// TIA Portal project "analog" (V17)
// Vorlageprojekt für das Buch mit Zielsystem S7-1200

(* hardware
DEVICE "S7-1200-Station_1"  S7-1200 Station
   slot 0: "Baugruppenträger_0"  Rack  V1.0
   slot 1: "PLC_1"  CPU 1211C DC/DC/DC  6ES7 211-1AE40-0XB0  V4.1
*)

// ===== PLC "PLC_1"  CPU 1211C DC/DC/DC =====

VAR_GLOBAL   // PLC tag table "Standard-Variablentabelle"
   "movingX" AT %I0.0 : Bool;
   "movingZ" AT %I0.1 : Bool;
   "itemDetected" AT %I0.2 : Bool;
   "lidAtPLace" AT %I0.3 : Bool;
   "lidClamped" AT %I0.4 : Bool;
   "PosAtLImit(Lids)" AT %I0.5 : Bool;
   "baseAtPlace" AT %I0.6 : Bool;
   "baseClamped" AT %I0.7 : Bool;
   "PosAtLImit(bases)" AT %I1.0 : Bool;
   "partLeaving" AT %I1.1 : Bool;
   "start" AT %I1.2 : Bool;
   "reset" AT %I1.3 : Bool;
   "stop" AT %I1.4 : Bool;
   "emergencyStop" AT %I1.5 : Bool;
   "auto" AT %I1.6 : Bool;
   "factoryIORunning" AT %I1.7 : Bool;
   "moveX" AT %Q0.0 : Bool;
   "moveZ" AT %Q0.1 : Bool;
   "grab" AT %Q0.2 : Bool;
   "lidsConveyor" AT %Q0.3 : Bool;
   "clampLid" AT %Q0.4 : Bool;
   "posRaise(lids)" AT %Q0.5 : Bool;
   "basesConveyor" AT %Q0.6 : Bool;
   "clampBAse" AT %Q0.7 : Bool;
   "posRaise(bases)" AT %Q1.0 : Bool;
   "startLight" AT %Q1.1 : Bool;
   "resetLight" AT %Q1.2 : Bool;
   "stopLight" AT %Q1.3 : Bool;
   "counter" AT %QD30 : DWord;
   "autoMode" AT %M0.0 : Bool;
   "manualMode" AT %M0.1 : Bool;
   "emergencyActivated" AT %M0.2 : Bool;
   "Clock_Byte" AT %MB10 : Byte;
   "Clock_10Hz" AT %M10.0 : Bool;
   "Clock_5Hz" AT %M10.1 : Bool;
   "Clock_2.5Hz" AT %M10.2 : Bool;
   "Clock_2Hz" AT %M10.3 : Bool;
   "Clock_1.25Hz" AT %M10.4 : Bool;
   "Clock_1Hz" AT %M10.5 : Bool;
   "Clock_0.625Hz" AT %M10.6 : Bool;
   "Clock_0.5Hz" AT %M10.7 : Bool;
   "systemRun" AT %M0.3 : Bool;
   "resetMode" AT %M0.4 : Bool;
   "Tag_1" AT %M8.0 : Bool;
   "Tag_2" AT %M8.1 : Bool;
   "Tag_3" AT %M8.2 : Bool;
   "lidAligned" AT %M0.5 : Bool;
   "moveZBit1" AT %M0.6 : Bool;
   "Tag_4" AT %M8.3 : Bool;
   "Tag_5" AT %M8.4 : Bool;
   "initiateStep8" AT %M0.7 : Bool;
   "Tag_6" AT %M8.5 : Bool;
   "Tag_7" AT %M8.6 : Bool;
   "moveZBit2" AT %M1.0 : Bool;
   "Tag_8" AT %M8.7 : Bool;
   "temp1" AT %M1.1 : Bool;
   "temp2" AT %M1.2 : Bool;
   "Tag_9" AT %M9.0 : Bool;
   "Tag_10" AT %M9.2 : Bool;
   "loop" AT %M1.3 : Bool;
END_VAR

DATA_BLOCK "manualCounterCount"   // DB4
{ S7_Optimized_Access := 'TRUE' }
VERSION : 0.1
   VAR
      manualCount : Int := -1;
   END_VAR
BEGIN
END_DATA_BLOCK

// folder: System blocks/Program resources

DATA_BLOCK "timer1"   // DB1
{ S7_Optimized_Access := 'TRUE' }
AUTHOR : Simatic
FAMILY : IEC
NAME : IEC_TMR
VERSION : 1.0
// stored: InstanceOfName IEC_TIMER
"IEC_TIMER"
BEGIN
END_DATA_BLOCK

DATA_BLOCK "timer2"   // DB2
{ S7_Optimized_Access := 'TRUE' }
AUTHOR : Simatic
FAMILY : IEC
NAME : IEC_TMR
VERSION : 1.0
// stored: InstanceOfName IEC_TIMER
"IEC_TIMER"
BEGIN
END_DATA_BLOCK

// folder: (top level)

FUNCTION "modesOf Operation" : Void   // FC1, LAD
{ S7_Optimized_Access := 'TRUE' }
VERSION : 0.1
   VAR_TEMP   // added for the SCL form of the ladder/FBD networks
      _w1 : Bool;
   END_VAR
BEGIN

REGION Network 1: Manual/AutoMode selector switch
   // Switches between manual and automatic modes
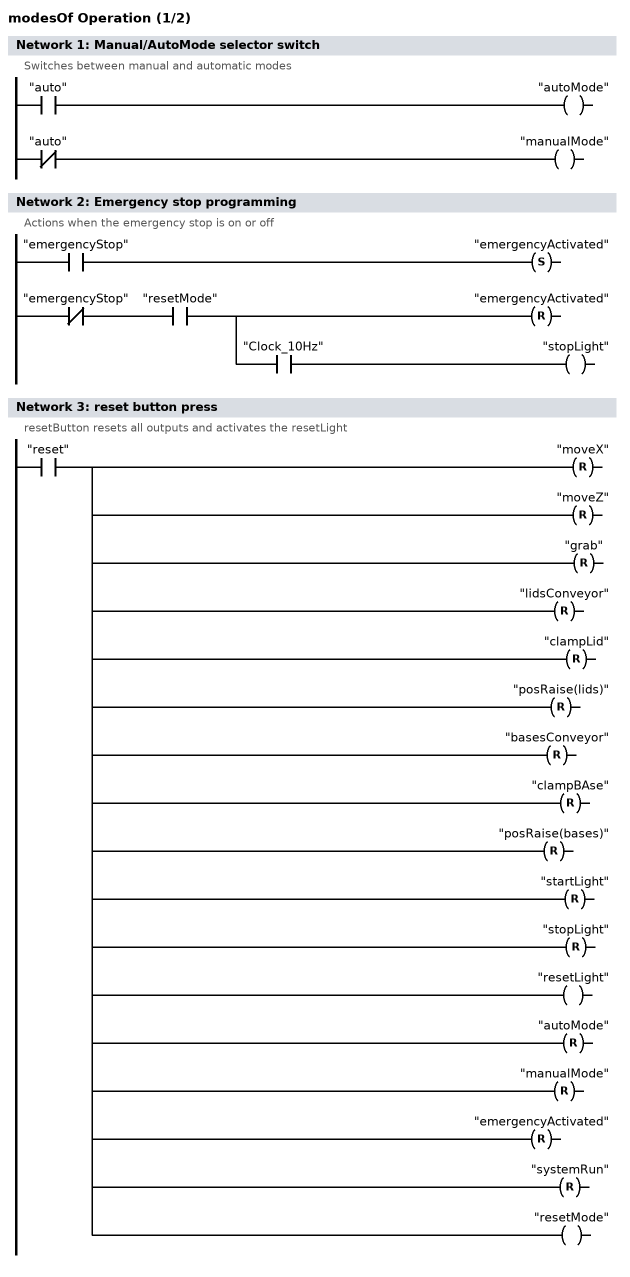
   RUNG wire#powerrail
      Contact( "auto" )
      Coil( "autoMode" )
   END_RUNG
   RUNG wire#powerrail
      I_Contact( "auto" )
      Coil( "manualMode" )
   END_RUNG
   // the same network as SCL:
   "autoMode" := "auto";
   "manualMode" := NOT "auto";
END_REGION

REGION Network 2: Emergency stop programming
   // Actions when the emergency stop is on or off
   RUNG wire#powerrail
      Contact( "emergencyStop" )
      S_Coil( "emergencyActivated" )
   END_RUNG
   RUNG wire#powerrail
      I_Contact( "emergencyStop" )
      Contact( "resetMode" )
      wire#w1
      R_Coil( "emergencyActivated" )
   END_RUNG
   RUNG wire#w1
      Contact( "Clock_10Hz" )
      Coil( "stopLight" )
   END_RUNG
   // the same network as SCL:
   IF "emergencyStop" THEN "emergencyActivated" := TRUE; END_IF;
   #_w1 := NOT "emergencyStop" AND "resetMode";
   IF #_w1 THEN "emergencyActivated" := FALSE; END_IF;
   "stopLight" := #_w1 AND "Clock_10Hz";
END_REGION

REGION Network 3: reset button press
   // resetButton resets all outputs and activates the resetLight
   RUNG wire#powerrail
      Contact( "reset" )
      wire#w1
      R_Coil( "moveX" )
   END_RUNG
   RUNG wire#w1
      R_Coil( "moveZ" )
   END_RUNG
   RUNG wire#w1
      R_Coil( "grab" )
   END_RUNG
   RUNG wire#w1
      R_Coil( "lidsConveyor" )
   END_RUNG
   RUNG wire#w1
      R_Coil( "clampLid" )
   END_RUNG
   RUNG wire#w1
      R_Coil( "posRaise(lids)" )
   END_RUNG
   RUNG wire#w1
      R_Coil( "basesConveyor" )
   END_RUNG
   RUNG wire#w1
      R_Coil( "clampBAse" )
   END_RUNG
   RUNG wire#w1
      R_Coil( "posRaise(bases)" )
   END_RUNG
   RUNG wire#w1
      R_Coil( "startLight" )
   END_RUNG
   RUNG wire#w1
      R_Coil( "stopLight" )
   END_RUNG
   RUNG wire#w1
      Coil( "resetLight" )
   END_RUNG
   RUNG wire#w1
      R_Coil( "autoMode" )
   END_RUNG
   RUNG wire#w1
      R_Coil( "manualMode" )
   END_RUNG
   RUNG wire#w1
      R_Coil( "emergencyActivated" )
   END_RUNG
   RUNG wire#w1
      R_Coil( "systemRun" )
   END_RUNG
   RUNG wire#w1
      Coil( "resetMode" )
   END_RUNG
   // the same network as SCL:
   IF "reset" THEN
       "moveX" := FALSE;
       "moveZ" := FALSE;
       "grab" := FALSE;
       "lidsConveyor" := FALSE;
       "clampLid" := FALSE;
       "posRaise(lids)" := FALSE;
       "basesConveyor" := FALSE;
       "clampBAse" := FALSE;
       "posRaise(bases)" := FALSE;
       "startLight" := FALSE;
       "stopLight" := FALSE;
   END_IF;
   "resetLight" := "reset";
   IF "reset" THEN
       "autoMode" := FALSE;
       "manualMode" := FALSE;
       "emergencyActivated" := FALSE;
       "systemRun" := FALSE;
   END_IF;
   "resetMode" := "reset";
END_REGION

REGION Network 4: Start button press
   // when the start button is pressed it should activate the system should run . Action of the stop and emergency stop should stop the system from working
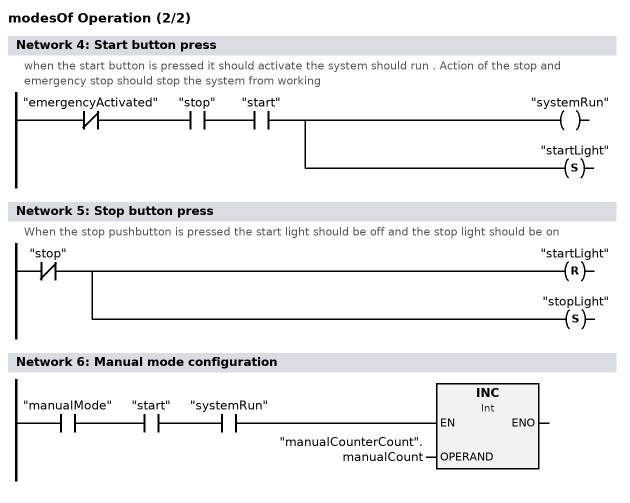
   RUNG wire#powerrail
      I_Contact( "emergencyActivated" )
      Contact( "stop" )
      Contact( "start" )
      wire#w1
      Coil( "systemRun" )
   END_RUNG
   RUNG wire#w1
      S_Coil( "startLight" )
   END_RUNG
   // the same network as SCL:
   "systemRun" := NOT "emergencyActivated" AND "stop" AND "start";
   IF "systemRun" THEN "startLight" := TRUE; END_IF;
END_REGION

REGION Network 5: Stop button press
   // When the stop pushbutton is pressed the start light should be off and the stop light should be on
   RUNG wire#powerrail
      I_Contact( "stop" )
      wire#w1
      R_Coil( "startLight" )
   END_RUNG
   RUNG wire#w1
      S_Coil( "stopLight" )
   END_RUNG
   // the same network as SCL:
   IF NOT "stop" THEN
       "startLight" := FALSE;
       "stopLight" := TRUE;
   END_IF;
END_REGION

REGION Network 6: Manual mode configuration
   RUNG wire#powerrail
      Contact( "manualMode" )
      Contact( "start" )
      Contact( "systemRun" )
      { S7_Templates := "DestType := Int" } Inc( "manualCounterCount".manualCount )
   END_RUNG
   // the same network as SCL:
   IF "manualMode" AND "start" AND "systemRun" THEN
       "manualCounterCount".manualCount := "manualCounterCount".manualCount + 1;
   END_IF;
END_REGION
END_FUNCTION

FUNCTION "stepDfn" : Void   // FC2, LAD
{ S7_Optimized_Access := 'TRUE' }
VERSION : 0.1
   VAR_TEMP   // added for the SCL form of the ladder/FBD networks
      _w1 : Bool;
      _w2 : Bool;
   END_VAR
BEGIN

REGION Network 1: Step 1
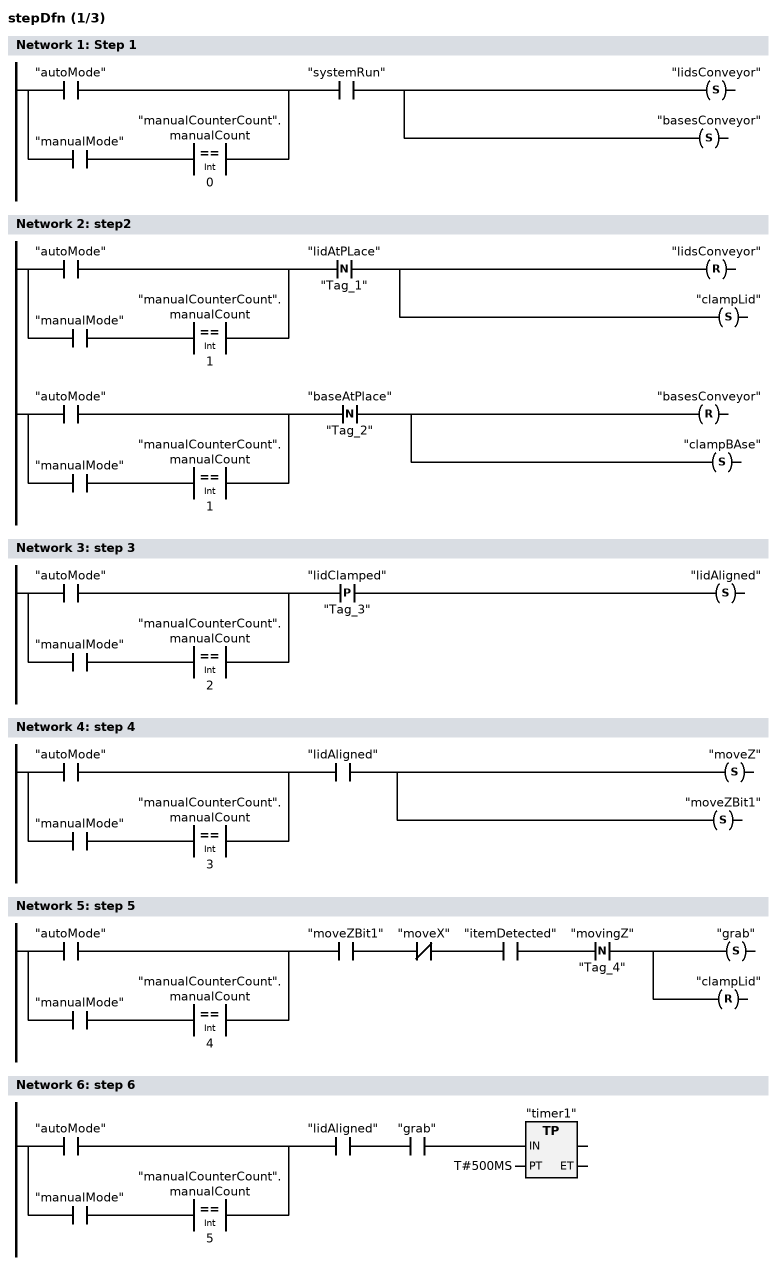
   RUNG wire#powerrail
      Contact( "autoMode" )
      wire#w1
      Contact( "systemRun" )
      wire#w2
      S_Coil( "lidsConveyor" )
   END_RUNG
   RUNG wire#powerrail
      Contact( "manualMode" )
      { S7_Templates := "SrcType := Int" } EQ_Contact(in1 := "manualCounterCount".manualCount, in2 := 0)
   END_RUNG wire#w1
   RUNG wire#w2
      S_Coil( "basesConveyor" )
   END_RUNG
   // the same network as SCL:
   IF ("autoMode" OR ("manualMode" AND ("manualCounterCount".manualCount = 0))) AND "systemRun" THEN
       "lidsConveyor" := TRUE;
       "basesConveyor" := TRUE;
   END_IF;
END_REGION

REGION Network 2: step2
   RUNG wire#powerrail
      Contact( "autoMode" )
      wire#w1
      N_Contact(operand := "lidAtPLace", bit := "Tag_1")
      wire#w2
      R_Coil( "lidsConveyor" )
   END_RUNG
   RUNG wire#powerrail
      Contact( "manualMode" )
      { S7_Templates := "SrcType := Int" } EQ_Contact(in1 := "manualCounterCount".manualCount, in2 := 1)
   END_RUNG wire#w1
   RUNG wire#w2
      S_Coil( "clampLid" )
   END_RUNG
   RUNG wire#powerrail
      Contact( "autoMode" )
      wire#w3
      N_Contact(operand := "baseAtPlace", bit := "Tag_2")
      wire#w4
      R_Coil( "basesConveyor" )
   END_RUNG
   RUNG wire#powerrail
      Contact( "manualMode" )
      { S7_Templates := "SrcType := Int" } EQ_Contact(in1 := "manualCounterCount".manualCount, in2 := 1)
   END_RUNG wire#w3
   RUNG wire#w4
      S_Coil( "clampBAse" )
   END_RUNG
   // the same network as SCL:
   #_w1 := ("autoMode" OR ("manualMode" AND ("manualCounterCount".manualCount = 1))) AND NOT "lidAtPLace" AND "Tag_1";   // falling edge of "lidAtPLace"
   "Tag_1" := "lidAtPLace";
   IF #_w1 THEN
       "lidsConveyor" := FALSE;
       "clampLid" := TRUE;
   END_IF;
   #_w2 := ("autoMode" OR ("manualMode" AND ("manualCounterCount".manualCount = 1))) AND NOT "baseAtPlace" AND "Tag_2";   // falling edge of "baseAtPlace"
   "Tag_2" := "baseAtPlace";
   IF #_w2 THEN
       "basesConveyor" := FALSE;
       "clampBAse" := TRUE;
   END_IF;
END_REGION

REGION Network 3: step 3
   RUNG wire#powerrail
      Contact( "autoMode" )
      wire#w1
      P_Contact(operand := "lidClamped", bit := "Tag_3")
      S_Coil( "lidAligned" )
   END_RUNG
   RUNG wire#powerrail
      Contact( "manualMode" )
      { S7_Templates := "SrcType := Int" } EQ_Contact(in1 := "manualCounterCount".manualCount, in2 := 2)
   END_RUNG wire#w1
   // the same network as SCL:
   #_w1 := ("autoMode" OR ("manualMode" AND ("manualCounterCount".manualCount = 2))) AND "lidClamped" AND NOT "Tag_3";   // rising edge of "lidClamped"
   "Tag_3" := "lidClamped";
   IF #_w1 THEN "lidAligned" := TRUE; END_IF;
END_REGION

REGION Network 4: step 4
   RUNG wire#powerrail
      Contact( "autoMode" )
      wire#w1
      Contact( "lidAligned" )
      wire#w2
      S_Coil( "moveZ" )
   END_RUNG
   RUNG wire#powerrail
      Contact( "manualMode" )
      { S7_Templates := "SrcType := Int" } EQ_Contact(in1 := "manualCounterCount".manualCount, in2 := 3)
   END_RUNG wire#w1
   RUNG wire#w2
      S_Coil( "moveZBit1" )
   END_RUNG
   // the same network as SCL:
   IF ("autoMode" OR ("manualMode" AND ("manualCounterCount".manualCount = 3))) AND "lidAligned" THEN
       "moveZ" := TRUE;
       "moveZBit1" := TRUE;
   END_IF;
END_REGION

REGION Network 5: step 5
   RUNG wire#powerrail
      Contact( "autoMode" )
      wire#w1
      Contact( "moveZBit1" )
      I_Contact( "moveX" )
      Contact( "itemDetected" )
      N_Contact(operand := "movingZ", bit := "Tag_4")
      wire#w2
      S_Coil( "grab" )
   END_RUNG
   RUNG wire#powerrail
      Contact( "manualMode" )
      { S7_Templates := "SrcType := Int" } EQ_Contact(in1 := "manualCounterCount".manualCount, in2 := 4)
   END_RUNG wire#w1
   RUNG wire#w2
      R_Coil( "clampLid" )
   END_RUNG
   // the same network as SCL:
   #_w1 := ("autoMode" OR ("manualMode" AND ("manualCounterCount".manualCount = 4))) AND "moveZBit1" AND NOT "moveX" AND "itemDetected" AND NOT "movingZ" AND "Tag_4";   // falling edge of "movingZ"
   "Tag_4" := "movingZ";
   IF #_w1 THEN
       "grab" := TRUE;
       "clampLid" := FALSE;
   END_IF;
END_REGION

REGION Network 6: step 6
   "timer1".TP(IN := ("autoMode" OR ("manualMode" AND ("manualCounterCount".manualCount = 5))) AND "lidAligned" AND "grab",
               PT := T#500MS);
END_REGION

REGION Network 7: step 7
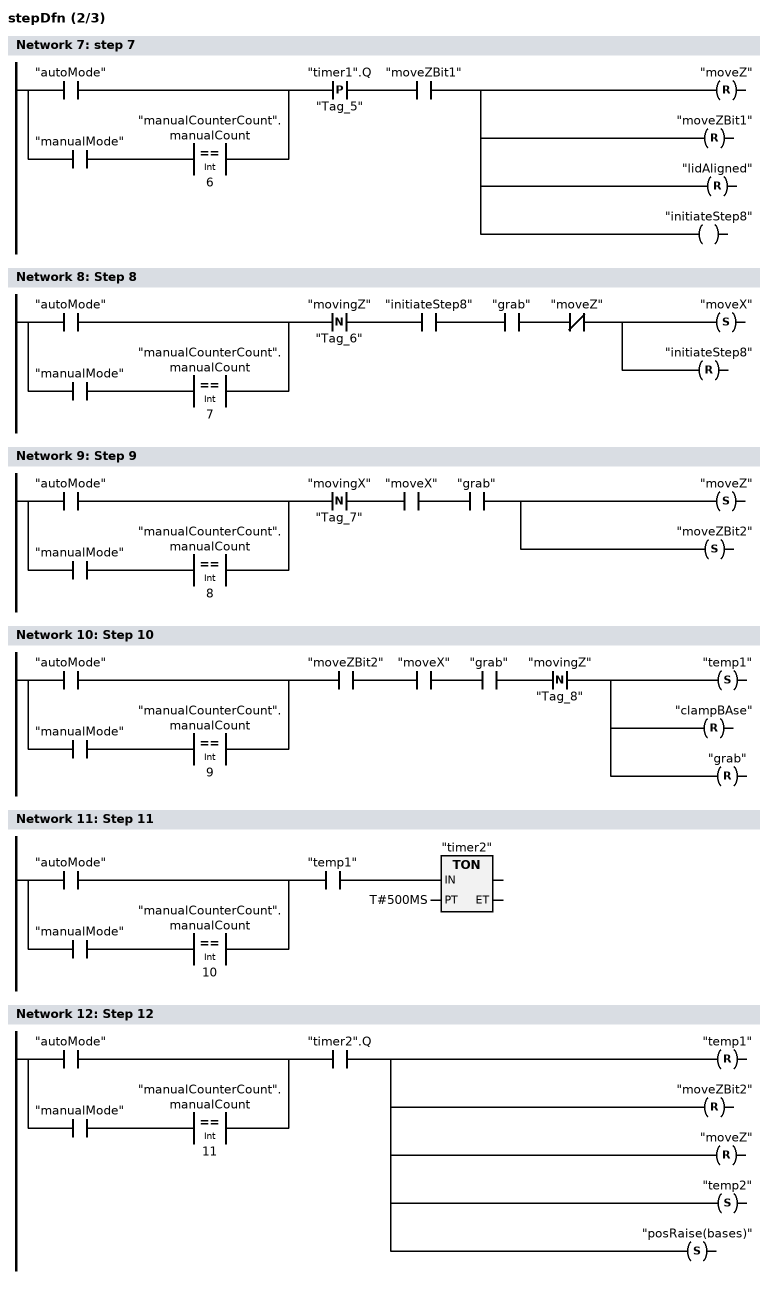
   RUNG wire#powerrail
      Contact( "autoMode" )
      wire#w1
      P_Contact(operand := "timer1".Q, bit := "Tag_5")
      Contact( "moveZBit1" )
      wire#w2
      R_Coil( "moveZ" )
   END_RUNG
   RUNG wire#powerrail
      Contact( "manualMode" )
      { S7_Templates := "SrcType := Int" } EQ_Contact(in1 := "manualCounterCount".manualCount, in2 := 6)
   END_RUNG wire#w1
   RUNG wire#w2
      R_Coil( "moveZBit1" )
   END_RUNG
   RUNG wire#w2
      R_Coil( "lidAligned" )
   END_RUNG
   RUNG wire#w2
      Coil( "initiateStep8" )
   END_RUNG
   // the same network as SCL:
   #_w1 := ("autoMode" OR ("manualMode" AND ("manualCounterCount".manualCount = 6))) AND "timer1".Q AND NOT "Tag_5";   // rising edge of "timer1".Q
   "Tag_5" := "timer1".Q;
   #_w2 := #_w1 AND "moveZBit1";
   IF #_w2 THEN
       "moveZ" := FALSE;
       "moveZBit1" := FALSE;
       "lidAligned" := FALSE;
   END_IF;
   "initiateStep8" := #_w2;
END_REGION

REGION Network 8: Step 8
   RUNG wire#powerrail
      Contact( "autoMode" )
      wire#w1
      N_Contact(operand := "movingZ", bit := "Tag_6")
      Contact( "initiateStep8" )
      Contact( "grab" )
      I_Contact( "moveZ" )
      wire#w2
      S_Coil( "moveX" )
   END_RUNG
   RUNG wire#powerrail
      Contact( "manualMode" )
      { S7_Templates := "SrcType := Int" } EQ_Contact(in1 := "manualCounterCount".manualCount, in2 := 7)
   END_RUNG wire#w1
   RUNG wire#w2
      R_Coil( "initiateStep8" )
   END_RUNG
   // the same network as SCL:
   #_w1 := ("autoMode" OR ("manualMode" AND ("manualCounterCount".manualCount = 7))) AND NOT "movingZ" AND "Tag_6";   // falling edge of "movingZ"
   "Tag_6" := "movingZ";
   IF #_w1 AND "initiateStep8" AND "grab" AND NOT "moveZ" THEN
       "moveX" := TRUE;
       "initiateStep8" := FALSE;
   END_IF;
END_REGION

REGION Network 9: Step 9
   RUNG wire#powerrail
      Contact( "autoMode" )
      wire#w1
      N_Contact(operand := "movingX", bit := "Tag_7")
      Contact( "moveX" )
      Contact( "grab" )
      wire#w2
      S_Coil( "moveZ" )
   END_RUNG
   RUNG wire#powerrail
      Contact( "manualMode" )
      { S7_Templates := "SrcType := Int" } EQ_Contact(in1 := "manualCounterCount".manualCount, in2 := 8)
   END_RUNG wire#w1
   RUNG wire#w2
      S_Coil( "moveZBit2" )
   END_RUNG
   // the same network as SCL:
   #_w1 := ("autoMode" OR ("manualMode" AND ("manualCounterCount".manualCount = 8))) AND NOT "movingX" AND "Tag_7";   // falling edge of "movingX"
   "Tag_7" := "movingX";
   IF #_w1 AND "moveX" AND "grab" THEN
       "moveZ" := TRUE;
       "moveZBit2" := TRUE;
   END_IF;
END_REGION

REGION Network 10: Step 10
   RUNG wire#powerrail
      Contact( "autoMode" )
      wire#w1
      Contact( "moveZBit2" )
      Contact( "moveX" )
      Contact( "grab" )
      N_Contact(operand := "movingZ", bit := "Tag_8")
      wire#w2
      S_Coil( "temp1" )
   END_RUNG
   RUNG wire#powerrail
      Contact( "manualMode" )
      { S7_Templates := "SrcType := Int" } EQ_Contact(in1 := "manualCounterCount".manualCount, in2 := 9)
   END_RUNG wire#w1
   RUNG wire#w2
      R_Coil( "clampBAse" )
   END_RUNG
   RUNG wire#w2
      R_Coil( "grab" )
   END_RUNG
   // the same network as SCL:
   #_w1 := ("autoMode" OR ("manualMode" AND ("manualCounterCount".manualCount = 9))) AND "moveZBit2" AND "moveX" AND "grab" AND NOT "movingZ" AND "Tag_8";   // falling edge of "movingZ"
   "Tag_8" := "movingZ";
   IF #_w1 THEN
       "temp1" := TRUE;
       "clampBAse" := FALSE;
       "grab" := FALSE;
   END_IF;
END_REGION

REGION Network 11: Step 11
   "timer2".TON(IN := ("autoMode" OR ("manualMode" AND ("manualCounterCount".manualCount = 10))) AND "temp1",
                PT := T#500MS);
END_REGION

REGION Network 12: Step 12
   RUNG wire#powerrail
      Contact( "autoMode" )
      wire#w1
      Contact( "timer2".Q )
      wire#w2
      R_Coil( "temp1" )
   END_RUNG
   RUNG wire#powerrail
      Contact( "manualMode" )
      { S7_Templates := "SrcType := Int" } EQ_Contact(in1 := "manualCounterCount".manualCount, in2 := 11)
   END_RUNG wire#w1
   RUNG wire#w2
      R_Coil( "moveZBit2" )
   END_RUNG
   RUNG wire#w2
      R_Coil( "moveZ" )
   END_RUNG
   RUNG wire#w2
      S_Coil( "temp2" )
   END_RUNG
   RUNG wire#w2
      S_Coil( "posRaise(bases)" )
   END_RUNG
   // the same network as SCL:
   IF ("autoMode" OR ("manualMode" AND ("manualCounterCount".manualCount = 11))) AND "timer2".Q THEN
       "temp1" := FALSE;
       "moveZBit2" := FALSE;
       "moveZ" := FALSE;
       "temp2" := TRUE;
       "posRaise(bases)" := TRUE;
   END_IF;
END_REGION

REGION Network 13: step 13
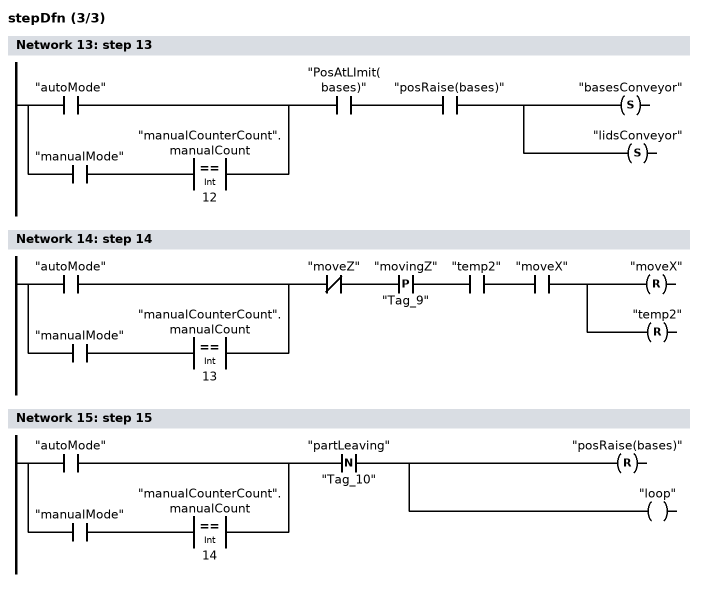
   RUNG wire#powerrail
      Contact( "autoMode" )
      wire#w1
      Contact( "PosAtLImit(bases)" )
      Contact( "posRaise(bases)" )
      wire#w2
      S_Coil( "basesConveyor" )
   END_RUNG
   RUNG wire#powerrail
      Contact( "manualMode" )
      { S7_Templates := "SrcType := Int" } EQ_Contact(in1 := "manualCounterCount".manualCount, in2 := 12)
   END_RUNG wire#w1
   RUNG wire#w2
      S_Coil( "lidsConveyor" )
   END_RUNG
   // the same network as SCL:
   IF ("autoMode" OR ("manualMode" AND ("manualCounterCount".manualCount = 12))) AND "PosAtLImit(bases)" AND "posRaise(bases)" THEN
       "basesConveyor" := TRUE;
       "lidsConveyor" := TRUE;
   END_IF;
END_REGION

REGION Network 14: step 14
   RUNG wire#powerrail
      Contact( "autoMode" )
      wire#w1
      I_Contact( "moveZ" )
      P_Contact(operand := "movingZ", bit := "Tag_9")
      Contact( "temp2" )
      Contact( "moveX" )
      wire#w2
      R_Coil( "moveX" )
   END_RUNG
   RUNG wire#powerrail
      Contact( "manualMode" )
      { S7_Templates := "SrcType := Int" } EQ_Contact(in1 := "manualCounterCount".manualCount, in2 := 13)
   END_RUNG wire#w1
   RUNG wire#w2
      R_Coil( "temp2" )
   END_RUNG
   // the same network as SCL:
   #_w1 := ("autoMode" OR ("manualMode" AND ("manualCounterCount".manualCount = 13))) AND NOT "moveZ" AND "movingZ" AND NOT "Tag_9";   // rising edge of "movingZ"
   "Tag_9" := "movingZ";
   #_w2 := #_w1 AND "temp2" AND "moveX";
   IF #_w2 THEN
       "moveX" := FALSE;
       "temp2" := FALSE;
   END_IF;
END_REGION

REGION Network 15: step 15
   RUNG wire#powerrail
      Contact( "autoMode" )
      wire#w1
      N_Contact(operand := "partLeaving", bit := "Tag_10")
      wire#w2
      R_Coil( "posRaise(bases)" )
   END_RUNG
   RUNG wire#powerrail
      Contact( "manualMode" )
      { S7_Templates := "SrcType := Int" } EQ_Contact(in1 := "manualCounterCount".manualCount, in2 := 14)
   END_RUNG wire#w1
   RUNG wire#w2
      Coil( "loop" )
   END_RUNG
   // the same network as SCL:
   #_w1 := ("autoMode" OR ("manualMode" AND ("manualCounterCount".manualCount = 14))) AND NOT "partLeaving" AND "Tag_10";   // falling edge of "partLeaving"
   "Tag_10" := "partLeaving";
   IF #_w1 THEN "posRaise(bases)" := FALSE; END_IF;
   "loop" := #_w1;
END_REGION
END_FUNCTION

FUNCTION "MHJ-PLC-Lab-Function-S71200" : Void   // FC9000, SCL
{ S7_Optimized_Access := 'TRUE' }
VERSION : 0.1
   VAR_TEMP
      rdTimeReturn : Int;
      outputTime : DTL;
      SyncVal : Byte;
      forVal : Int;
      forVal_2 : Int;
      Value : Byte;
   END_VAR
   VAR CONSTANT
      CompVal : Byte := 16#34;
      Value_01 : Byte := 16#11;
      Value_01_DW : DWord := 16#A165_D992;
      Value_02_DW : DWord := 16#58BE_4401;
   END_VAR
BEGIN

   #Value:=PEEK(area := 16#82,
        dbNumber := 0,
        byteOffset := 511);
   #Value := #Value + 1;

   POKE(area := 16#82,
        dbNumber := 0,
        byteOffset := 511,
        value := #Value);

   POKE(area:=16#81,
        dbNumber:=0,
        byteOffset:=1016,
        value:=#Value_01_DW);
   POKE(area := 16#81,
        dbNumber := 0,
        byteOffset := 1020,
        value := #Value_02_DW);

   POKE(area := 16#81,
        dbNumber := 0,
        byteOffset := 511,
        value := B#16#00);

   FOR #forVal := 0 TO 120 DO
       FOR #forVal_2:=0 TO 10 DO
           #rdTimeReturn:=RD_SYS_T(#outputTime);
           #rdTimeReturn := WR_SYS_T(#outputTime);
           #rdTimeReturn := RD_SYS_T(#outputTime);
           #rdTimeReturn := WR_SYS_T(#outputTime);
       END_FOR;
       #SyncVal:= PEEK(area := 16#81,
                      dbNumber := 0,
                      byteOffset := 511);
       IF #SyncVal = #CompVal THEN
          GOTO M_1;
       END_IF;
   END_FOR;
   RETURN;

   M_1:
   POKE(area := 16#81,
        dbNumber := 0,
        byteOffset := 511,
        value := B#16#0);
END_FUNCTION

ORGANIZATION_BLOCK "Main"   // OB1, LAD, ProgramCycle
TITLE = "Main Program Sweep (Cycle)"
{ S7_Optimized_Access := 'TRUE' }
VERSION : 0.1
   VAR_INPUT
      Initial_Call : Bool;   // Initial call of this OB
      Remanence : Bool;   // =True, if remanent data are available
   END_VAR
BEGIN

REGION Network 1: Konnektierungsbaustein für PLC-Lab
   // Im Netzwerk 1 wird der Konnektierungsbaustein für PLC-Lab aufgerufen.
   // Dieser Aufruf darf nicht entfernt werden!
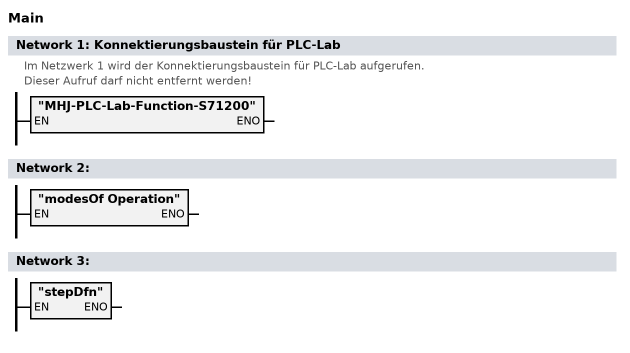
   RUNG wire#powerrail
      "MHJ-PLC-Lab-Function-S71200"()
   END_RUNG
   // the same network as SCL:
   "MHJ-PLC-Lab-Function-S71200"();
END_REGION

REGION Network 2
   RUNG wire#powerrail
      "modesOf Operation"()
   END_RUNG
   // the same network as SCL:
   "modesOf Operation"();
END_REGION

REGION Network 3
   RUNG wire#powerrail
      "stepDfn"()
   END_RUNG
   // the same network as SCL:
   "stepDfn"();
END_REGION
END_ORGANIZATION_BLOCK